TYPE OperationLimits :
STRUCT
	rMinPosition		:		REAL;
	rMaxPosition		:		REAL;
	rMaxVelocity		:		REAL;
	rJogVelocity		:		REAL;
	tMaxMotionTime		:		TIME;
END_STRUCT
END_TYPE

(* stored: Version 1.1.0.1, ProductVersion 3.1.4024.6
   DUT OperationLimits: Id {7418df94-aee6-4511-973c-934c4f785c97} *)
